	999: //Group Reset Error
		_Error				:= _PlanarFb.Error;
		_ErrorID			:= _PlanarFb.ErrorId;
		_BlockingObjectInfo := _PlanarFb.objectInfo;
END_CASE

Execute := THIS^;

//Heartbeat that the method is active
ExecuteWatchdog := ExecuteWatchdog + 1;
END_METHOD

METHOD Update
VAR_INST
	WatchdogCheck : UDINT;
END_VAR
IF ExecuteWatchdog <> WatchdogCheck THEN
	WatchdogCheck := ExecuteWatchdog;
ELSE
	HasRun			:= FALSE;
	TaskState		:= 0;
	ExecuteWatchdog := 0;
END_IF

_PlanarFb.Update();
THIS^.Busy := TaskState > 0 AND TaskState < 50;
END_METHOD

END_FUNCTION_BLOCK

// XPlanarComponent/FB_Component_XPlanar
{attribute 'no_assign'}
{attribute 'no_explicit_call' := 'do not call this POU directly'}
FUNCTION_BLOCK FB_Component_XPlanar EXTENDS FB_ComponentBase
VAR
	Parts			  : ARRAY[1..Param_TcIoXPlanarEnvironment.MaxParts] OF FB_XPlanarPart;
	Tiles			  : ARRAY[1..Param_TcIoXPlanarEnvironment.MaxTiles] OF FB_XPlanarTile;
	ipMoverCyclic	  : ARRAY[1..SystemParameters.MOVER_COUNT] OF I_CyclicFB;
	ipTrackCyclic	  : ARRAY[1..SystemParameters.TRACK_COUNT] OF I_CyclicFB;
	UtilityVisu		  : FB_XPlanarUtilityVisu;

	//System Level Tasks
	EnablePlanarGroup	: FB_EnableGroup;
	MoverDetection		: FB_MoverRedetection;
	MoverIdentification : FB_MoverIdentification;
	XPlanarReset		: FB_ResetXPlanar;

	//Helper Vars
	_OperationMode		: XPlanarOperationMode;
	_Xpu				: I_TcIoXPlanarProcessingUnit;
	_TracksInitialized	: BOOL;
	_MoverDetectionInfo : ST_TcIoMoverDetectionInfos;
	AbortState			: UDINT;
END_VAR

//! Provides basic error detection and event handling for this component
METHOD PROTECTED Monitoring
(*! @descriptionThis method is called cyclically by <c>CyclicLogic()</c>*)
VAR
	i	   : UDINT;
	Result : HRESULT;
END_VAR
//Watch for mover error
FOR i := 1 TO SystemParameters.MOVER_COUNT DO
	IF ip.Movers[i].Error THEN
		_Error	 := TRUE;
		_ErrorID := ip.Movers[i].ErrorID;
		EXIT;
	END_IF
END_FOR

//Watch for Track Error
FOR i := 1 TO SystemParameters.TRACK_COUNT DO
	IF ip.Tracks[i].Error THEN
		_Error := TRUE;
		_ErrorID := ip.Tracks[i].ErrorID;
		EXIT;
	END_IF
END_FOR

IF _Error THEN
	_CurrentAlarmSeverity := TcEventSeverity.Error;
END_IF
END_METHOD

//! @summary This method serves as the entry point for all underlying FB logic
METHOD PUBLIC CyclicLogic
//! @description This method should be called cyclically by descendant function blocks by invoking <c>SUPER^.CyclicLogic()</c>.  Alternatively, the contents of this method could be reimplemented entirely in which case a call to this method would not be necessary.
VAR_Inst
	i : UDINT;
END_VAR
//Update Xplanar system status
XPlanar.Environment.Update();
XPlanar.Group.Update();

//Update Internal Mover state - Must be called every cycle 
FOR i := 1 TO SystemParameters.MOVER_COUNT DO
	IF ip.Movers[i] <> 0 THEN
		ip.Movers[i].pm.Update();
	END_IF
END_FOR

//Update INTERNAL Track status - Must be called every cycle 
FOR i := 1 TO SystemParameters.TRACK_COUNT DO
	IF ip.Tracks[i] <> 0 THEN
		ip.Tracks[i].pm.Update();
	END_IF
END_FOR

EnablePlanarGroup.Update();
MoverDetection.Update();
MoverIdentification.Update();
XPlanarReset.Update();

FOR i := 1 TO XPlanar.PartCount DO
	Parts[i].CyclicLogic();
END_FOR

//Make sure things are initialized
IF NOT _InitComplete THEN
	_InitComplete := Initialize();
	RETURN;
END_IF

//Update Mover status
FOR i := 1 TO SystemParameters.MOVER_COUNT DO
	IF ipMoverCyclic[i] <> 0 THEN
		ipMoverCyclic[i].CyclicLogic();
	END_IF
END_FOR

//Update Track status 
FOR i := 1 TO SystemParameters.TRACK_COUNT DO
	IF ipTrackCyclic[i] <> 0 THEN
		ipTrackCyclic[i].CyclicLogic();
	END_IF
END_FOR

//Update Station IDs
FOR i := 1 TO SystemParameters.STATION_COUNT DO
	IF ip.Stations[i] <> 0 THEN
		ip.Stations[i].ID := i;
	END_IF
END_FOR

FOR i := 1 TO XPlanar.TileCount DO
	Tiles[i].CyclicLogic();
END_FOR

//Update Utility Visu
UtilityVisu.Cycle();
SUPER^.CyclicLogic();
END_METHOD

METHOD Abort : BOOL
VAR
	i	   : UDINT := 1;
	Result : BOOL;
END_VAR

VAR_INST
	MoversHalted   : BOOL;
	MoversDisabled : BOOL;
	TracksDisabled : BOOL;
	ErrString	   : STRING;
END_VAR
CASE AbortState OF
	0:
		AbortState := AbortState + 10;

	10: //Halt System
		FOR i := 1 TO SystemParameters.MOVER_COUNT DO
			ip.Movers[i].Halt();
		END_FOR

		AbortState := AbortState + 10;

	20: //Monitor Halt System Feedback
		MoversHalted := TRUE;
		FOR i := 1 TO SystemParameters.MOVER_COUNT DO
			IF ip.Movers[i].Status.Busy.busyMover AND (ip.Movers[i].Status.State <> Mc_Planar_State.Error) THEN
				MoversHalted := FALSE;
			END_IF
		END_FOR

		IF MoversHalted THEN
			AbortState := AbortState + 10;
		END_IF

	30: //Disable Movers
		FOR i := 1 TO SystemParameters.MOVER_COUNT DO
			ip.Movers[i].Disable();
		END_FOR

		AbortState := AbortState + 10;

	40: //Check disable command feedback
		MoversDisabled := TRUE;
		FOR i := 1 TO SystemParameters.MOVER_COUNT DO
			IF (ip.Movers[i].Status.State <> Mc_Planar_State.Disabled) AND (ip.Movers[i].Status.State <> Mc_Planar_State.Error) THEN
				MoversDisabled := FALSE;
			END_IF
		END_FOR

		IF MoversDisabled THEN
			AbortState := AbortState + 10;
		END_IF

	50: //Disable Tracks
		FOR i := 1 TO SystemParameters.TRACK_COUNT DO
			ip.Tracks[i].Disable();
		END_FOR

		AbortState := AbortState + 10;

	60: //Monitor track disable feedback
		TracksDisabled := TRUE;
		FOR i := 1 TO SystemParameters.TRACK_COUNT DO
			IF (ip.Tracks[i].Status.State <> Mc_Planar_State.Disabled) AND (ip.Tracks[i].Status.State <> Mc_Planar_State.Error) THEN
				MoversDisabled := FALSE;
			END_IF
		END_FOR

		AbortState := AbortState + 10;

	70: //Make sure sequences are reset
		AbortState := AbortState + 10;

	80: //Abort Complete	
		Abort	   := TRUE;
		AbortState := 0;

	999: //Error
		Abort	   := TRUE;
		AbortState := 0;
		_Error	   := TRUE;
END_CASE
END_METHOD

METHOD AddMoversToGroup : I_PlanarTaskResult
VAR_INST
	i			   : UDINT;
	Result		   : FB_ResultBase;
	AddGroupResult : I_PlanarTaskResult;
	MoversInGroup  : BOOL;
END_VAR
MoversInGroup  := FALSE;
Result.Busy	   := TRUE;
Result.Done	   := FALSE;
Result.Error   := FALSE;
Result.ErrorID := 0;
FOR i := 1 TO SystemParameters.MOVER_COUNT DO
	AddGroupResult := ip.Movers[i].AddToGroup(XPlanar.Group);
	IF AddGroupResult.Error THEN
		Result.Error   := AddGroupResult.Error;
		Result.ErrorID := AddGroupResult.ErrorID;
		Result.Busy	   := FALSE;
		EXIT;
	END_IF
END_FOR

MoversInGroup := TRUE;
FOR i := 1 TO SystemParameters.MOVER_COUNT DO
	IF ip.Movers[i].Status.GroupOID = 0 THEN
		MoversInGroup := FALSE;
	END_IF
END_FOR

IF MoversInGroup THEN
	Result.Busy := FALSE;
	Result.Done := TRUE;
END_IF

AddMoversToGroup := Result;
END_METHOD

METHOD AddTracksToGroup : I_PlanarTaskResult
VAR_INST
	i			   : UDINT;
	AddGroupResult : I_PlanarTaskResult;
	Result		   : FB_ResultBase;
	TracksInGroup  : BOOL;
END_VAR
TracksInGroup  := FALSE;
Result.Busy	   := TRUE;
Result.Done	   := FALSE;
Result.Error   := FALSE;
Result.ErrorID := 0;
FOR i := 1 TO SystemParameters.TRACK_COUNT DO
	AddGroupResult := ip.Tracks[i].AddToGroup(XPlanar.Group);
	IF AddGroupResult.Error THEN
		Result.Error   := AddGroupResult.Error;
		Result.ErrorID := AddGroupResult.ErrorID;
		Result.Busy	   := FALSE;
		EXIT;
	END_IF
END_FOR

TracksInGroup := TRUE;
FOR i := 1 TO SystemParameters.TRACK_COUNT DO
	IF ip.Tracks[i].Status.GroupOID = 0 THEN
		TracksInGroup := FALSE;
	END_IF
END_FOR

IF TracksInGroup THEN
	Result.Busy := FALSE;
	Result.Done := TRUE;
END_IF

AddTracksToGroup := Result;
END_METHOD

METHOD DisableMovers : I_PlanarTaskResult
VAR_INST
	i			   : UDINT := 1;
	j			   : UDINT := 1;
	MoversDisabled : BOOL;
	CommandResult  : I_PlanarTaskResult;
	Result		   : FB_ResultBase;
END_VAR
Result.Done	   := FALSE;
Result.Error   := FALSE;
Result.ErrorID := 0;
IF i <= SystemParameters.MOVER_COUNT THEN
	CommandResult := ip.Movers[i].Disable();
	IF CommandResult.Done THEN
		i := i + 1;
	ELSIF CommandResult.Error THEN
		_ErrorID	   := CommandResult.ErrorID;
		Result.Error   := CommandResult.Error;
		Result.ErrorID := CommandResult.ErrorID;
//		RaiseAlarmWithStrings(Alarm := XPlanarBaseAlarms[E_XPlanarApplicationEventClass.SystemError], CONCAT('Mover ', TO_STRING(i)), CONCAT('EnableError ', TO_STRING(_ErrorID)));
	END_IF
ELSE
	i := 1;
END_IF

MoversDisabled := TRUE;
FOR j := 1 TO SystemParameters.MOVER_COUNT DO
	IF ip.Movers[j].Status.State = Mc_Planar_State.Enabled THEN
		MoversDisabled := FALSE;
	END_IF
END_FOR

IF MoversDisabled THEN
	Result.Done := TRUE;
END_IF

DisableMovers := Result;
END_METHOD

METHOD EnableGroup : I_PlanarTaskResult
EnableGroup := EnablePlanarGroup.Execute();
END_METHOD

METHOD EnableMovers : I_PlanarTaskResult
VAR_INST
	i			  : UDINT := 1;
	j			  : UDINT := 1;
	MoversEnabled : BOOL;
	EnableResult  : I_PlanarTaskResult;
	Result		  : FB_ResultBase;
END_VAR
Result.Done	   := FALSE;
Result.Error   := FALSE;
Result.ErrorID := 0;
IF i <= SystemParameters.MOVER_COUNT THEN
	EnableResult := ip.Movers[i].Enable();
	IF EnableResult.Done THEN
		i := i + 1;
	ELSIF EnableResult.Error THEN
		_ErrorID	   := EnableResult.ErrorID;
		Result.Error   := EnableResult.Error;
		Result.ErrorID := EnableResult.ErrorID;
	END_IF
ELSE
	i := 1;
END_IF

MoversEnabled := TRUE;
FOR j := 1 TO SystemParameters.MOVER_COUNT DO
	IF ip.Movers[j].Status.State <> Mc_Planar_State.Enabled THEN
		MoversEnabled := FALSE;
	END_IF
END_FOR

IF MoversEnabled THEN
	Result.Done := TRUE;
END_IF

EnableMovers := Result;
END_METHOD

METHOD EnableTracks : I_PlanarTaskResult
VAR_INST
	i			  : UDINT := 1;
	j			  : UDINT := 1;
	TracksEnabled : BOOL;
	Result		  : FB_ResultBase;
	EnableResult  : I_PlanarTaskResult;
END_VAR
Result.Done	   := FALSE;
Result.Error   := FALSE;
Result.ErrorID := 0;
IF i <= SystemParameters.TRACK_COUNT THEN
	EnableResult := ip.Tracks[i].Enable();
	IF EnableResult.Done THEN
		i := i + 1;
	ELSIF EnableResult.Error THEN
		_ErrorID	   := EnableResult.ErrorID;
		Result.Error   := EnableResult.Error;
		Result.ErrorID := EnableResult.ErrorID;
	END_IF
ELSE
	i := 1;
END_IF

TracksEnabled := TRUE;
FOR j := 1 TO SystemParameters.TRACK_COUNT DO
	IF ip.Tracks[j].Status.State <> Mc_Planar_State.Enabled THEN
		TracksEnabled := FALSE;
	END_IF
END_FOR

IF TracksEnabled THEN
	Result.Done := TRUE;
END_IF

EnableTracks := Result;
END_METHOD

METHOD IdentifyMovers : I_PlanarTaskResult
VAR
	Result : BOOL;
END_VAR

VAR_INST
	IdentificationStatus : Tc3_XplanarUtility.MoverIdentificationStatus;
END_VAR
IdentifyMovers := MoverIdentification.Execute();
END_METHOD

//! @summary Basic component initialization logic
METHOD PROTECTED Initialize : BOOL;
//! @description This method is called by <c>CyclicLogic()</c> as required
VAR_INST
	i			   : UINT;
	SequenceState  : UDINT;
	TrackToInit	   : UDINT := 1;
	TilePosition   : ST_TcIoTilePositionOnPart;
	MoverType	   : XPlanarMoverType;
	InitPartResult : I_PlanarTaskResult;
END_VAR
Initialize := FALSE;
CASE SequenceState OF
	0: //Init
		IF SUPER^.Initialize() THEN
			SequenceState := SequenceState + 10;
		END_IF

	10: //Init XPlanar Environment
		IF Xplanar.EnvironmentTcIo.Init(TRUE) THEN
			Xplanar.EnvironmentTcIo.Init(FALSE);
			SequenceState := SequenceState + 10;
		ELSIF Xplanar.EnvironmentTcIo.Error THEN
			RETURN;
		END_IF

	20: //Get Operation Mode
		XPlanar.OperationMode := XPlanar.EnvironmentTcIo.TcIoXpu(1).GetOperationMode();
		SequenceState		  := SequenceState + 10;

	30: //Get XPU OIDs
		IF XPlanar.EnvironmentTcIo.P_XpuCount > 0 THEN
			IF XPlanar.EnvironmentTcIo.GetXpuOids(TRUE) THEN
				XPlanar.EnvironmentTcIo.GetXpuOids(FALSE);
				SequenceState := SequenceState + 10;
			ELSIF Xplanar.EnvironmentTcIo.Error THEN
				SequenceState := 999;
			END_IF;
		END_IF

	40: //Set XPU Interfaces
		_Xpu					:= XPlanar.EnvironmentTcIo.TcIoXpu(1);
		UtilityVisu.Environment := XPlanar.EnvironmentTcIo;
		SequenceState			:= SequenceState + 10;

	50: //Get Part OIDs
		XPlanar.PartCount := TO_UINT(_Xpu.GetPartCount());
		IF _Xpu.GetPartOids() THEN
			SequenceState := SequenceState + 10;
		END_IF

	60: //Assign OIDs to Part Objects
		IF XPlanar.PartCount > 0 THEN
			FOR i := 1 TO XPlanar.PartCount DO
				Parts[i].ObjectID := _Xpu.P_PartOids[i];
			END_FOR
		END_IF

		i			  := 1;
		SequenceState := SequenceState + 10;

	70: //Initialize Parts
		IF i > 0 AND i <= XPlanar.PartCount THEN
			InitPartResult := Parts[i].Initialize();
			IF InitPartResult.Done THEN
				SequenceState := SequenceState + 1;
			ELSIF InitPartResult.Error THEN
				SequenceState := 999;
			END_IF
		ELSE
			i			  := 1;
			SequenceState := SequenceState + 10;
		END_IF

	71: //Loop back for next part
		i			  := i + 1;
		SequenceState := SequenceState - 1;

	80: //Set mover index values
		FOR i := 1 TO SystemParameters.MOVER_COUNT DO
			IF ip.Movers[i] <> 0 THEN
				__QUERYINTERFACE(ip.Movers[i], ipMoverCyclic[i]);
				ip.Movers[i].Utility	:= _Xpu.TcIoMover(TO_UINT(i));
				ip.Movers[i].MoverIndex := i;

				//Set initial mover dynamics
				ip.Movers[i].Dynamics.Movement.Accel	:= 2000;
				ip.Movers[i].Dynamics.Movement.Decel	:= 2000;
				ip.Movers[i].Dynamics.Movement.Velocity := 200;
				ip.Movers[i].Dynamics.Movement.Jerk		:= 50000;
				ip.Movers[i].Dynamics.Rotation.Accel	:= 5000;
				ip.Movers[i].Dynamics.Rotation.Decel	:= 5000;
				ip.Movers[i].Dynamics.Rotation.Velocity := 100;
				ip.Movers[i].Dynamics.Rotation.Jerk		:= 50000;
				ip.Movers[i].Dynamics.Tilt.Accel		:= 5000;
				ip.Movers[i].Dynamics.Tilt.Decel		:= 5000;
				ip.Movers[i].Dynamics.Tilt.Velocity		:= 200;
				ip.Movers[i].Dynamics.Tilt.Jerk			:= 50000;
			END_IF
		END_FOR

		XPlanar.MoverCount := SystemParameters.MOVER_COUNT;
		SequenceState	   := SequenceState + 10;

	90: //Set track index values
		FOR i := 1 TO SystemParameters.TRACK_COUNT DO
			__QUERYINTERFACE(ip.Tracks[i], ipTrackCyclic[i]);
			IF ip.Tracks[i] <> 0 THEN
				ip.Tracks[i].Index := i;
			END_IF
		END_FOR

		SequenceState := SequenceState + 10;

	100: //Get Tile Count
		XPlanar.TileCount := TO_UINT(XPlanar.EnvironmentTcIo.TcIoXpu(1).GetTileCount());
		i				  := 1;
		SequenceState	  := SequenceState + 10;

	110: //Initialize Tile Objects
		FOR i := 1 TO XPlanar.TileCount DO
			Tiles[i].Index := i;
			Tiles[i].Initialize();
		END_FOR

		FOR i := 1 TO XPlanar.MoverCount DO
			XPlanarHMI.MoverObjects[i].MoverBTN := XPlanar.EnvironmentTcIo.TcIoXpu(1).TcIoMover(i).GetBtn();
			MoverType							:= XPlanar.EnvironmentTcIo.TcIoXpu(1).TcIoMover(i).GetMoverType();
			IF MoverType = XPlanarMoverType.APM4220 THEN
				XPlanarHMI.MoverObjects[i].Width  := 115;
				XPlanarHMI.MoverObjects[i].Height := 115;
			ELSIF MoverType = XPlanarMoverType.APM4221 THEN
				XPlanarHMI.MoverObjects[i].Width  := 127;
				XPlanarHMI.MoverObjects[i].Height := 127;
			ELSIF MoverType = XPlanarMoverType.APM4330 THEN
				XPlanarHMI.MoverObjects[i].Width  := 155;
				XPlanarHMI.MoverObjects[i].Height := 155;
			ELSIF MoverType = XPlanarMoverType.APM4550 THEN
				XPlanarHMI.MoverObjects[i].Width  := 235;
				XPlanarHMI.MoverObjects[i].Height := 235;
			END_IF

			IF ip.Movers[i] <> 0 THEN
				ip.Movers[i].MoverType := MoverType;
			END_IF
		END_FOR

		SequenceState := SequenceState + 10;

	111:
		IF i < XPlanar.TileCount THEN
			i			  := 1 + 1;
			SequenceState := 80;
		ELSE
			i			  := 1;
			SequenceState := 90;
		END_IF

	120: //Init Complete
		Initialize := TRUE;

	999: // Init Error
		_Error	 := TRUE;
		_ErrorID := 9990;
		RETURN;
END_CASE
END_METHOD

{attribute 'suppress_wrn_C0410'}
PROPERTY MoverDetectionInfo : REFERENCE TO ST_TcIoMoverDetectionInfos
GET
MoverDetectionInfo ref= _MoverDetectionInfo;
END_GET
END_PROPERTY

METHOD MoverRedetect : I_PlanarTaskResult
VAR
	Result : BOOL;
END_VAR
MoverRedetect := MoverDetection.Execute();
END_METHOD

//! @summary Clears error flags and error IDs for this component
METHOD PUBLIC Reset : BOOL
VAR
	i : UDINT;
END_VAR

VAR_INST
	CommandResult : I_PlanarTaskResult;
END_VAR
CommandResult := XPlanarReset.Execute();

IF CommandResult.Done THEN
	_Error	 := FALSE;
	_ErrorID := 0;
	_CurrentAlarmSeverity := TcEventSeverity.Verbose;
	Reset	 := TRUE;
ELSIF CommandResult.Error THEN
	_Error := TRUE;
	_ErrorID := CommandResult.ErrorID;
END_IF
END_METHOD

PROPERTY TileCount : UDINT
GET
(*IF XPlanarSystem.ipDriver <> 0 THEN
	IF XPlanarSystem.ipDriver.XpuTcIo(1).GetOperationMode() = 0 THEN
		TileCount := XPlanarSystem.ipDriver.XpuTcIo(1).GetTileCount();
	END_IF
ELSE
	TileCount := 0; ///Marc TODO: What to return if the interface is not good?
END_IF
*)
END_GET
END_PROPERTY

PROPERTY TracksInitialized : BOOL
GET
TracksInitialized := _TracksInitialized;
END_GET
END_PROPERTY

PROPERTY Utility : I_TcIoXPlanarProcessingUnit
GET
Utility := _Xpu;
END_GET
END_PROPERTY

END_FUNCTION_BLOCK
